# EPICS StreamDevice protocol: PMD90Sup/devPMD90.proto
Separator = CR;
ExtraInput = Ignore;

valid_chars = "[a-zA-Z0-9._: ]";

read_float {
    @mismatch { in "!%(\$1ERROR_CODE)d"; }
    out "\$2?";
    in "%f";
}

set_float {
    @mismatch { in "!%(\$1ERROR_CODE)d"; }
    out "\$2 %f";
    in "!0";
}

# Generic
write {
    out "\$2";
}

write_int {
    out "\$2%d";
}

read_int {
    out "\$2";
    in "\$2 %d";
}

read_plain_int {
    out "\$2";
    in "%d";
}

read_string {
    out "\$2";
    in "%#s";
    InTerminator = "\r";
}
